// Mitsubishi GX Works2 project: Step Control   PLC: Q01U

PROGRAM conveyor
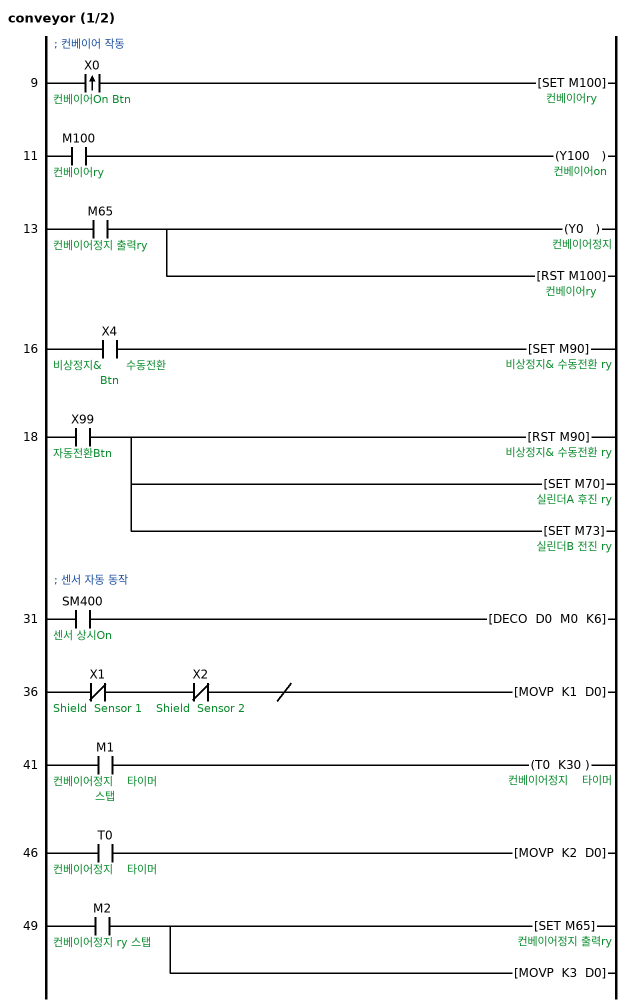
; 컨베이어 작동
9     LDP     X0  ; 컨베이어On Btn
      SET     M100  ; 컨베이어ry
11    LD      M100  ; 컨베이어ry
      OUT     Y100  ; 컨베이어on
13    LD      M65  ; 컨베이어정지 출력ry
      OUT     Y0  ; 컨베이어정지
      RST     M100  ; 컨베이어ry
16    LD      X4  ; 비상정지&       수동전환 Btn
      SET     M90  ; 비상정지& 수동전환 ry
18    LD      X99  ; 자동전환Btn
      RST     M90  ; 비상정지& 수동전환 ry
      SET     M70  ; 실린더A 후진 ry
      SET     M73  ; 실린더B 전진 ry
; 센서 자동 동작
31    LD      SM400  ; 센서 상시On
      DECO    D0 M0 K6
36    LDI     X1  ; Shield  Sensor 1
      ANI     X2  ; Shield  Sensor 2
      INV
      MOVP    K1 D0
41    LD      M1  ; 컨베이어정지    타이머  스탭
      OUT     T0 K30  ; 컨베이어정지    타이머
46    LD      T0  ; 컨베이어정지    타이머
      MOVP    K2 D0
49    LD      M2  ; 컨베이어정지 ry 스탭
      SET     M65  ; 컨베이어정지 출력ry
      MOVP    K3 D0
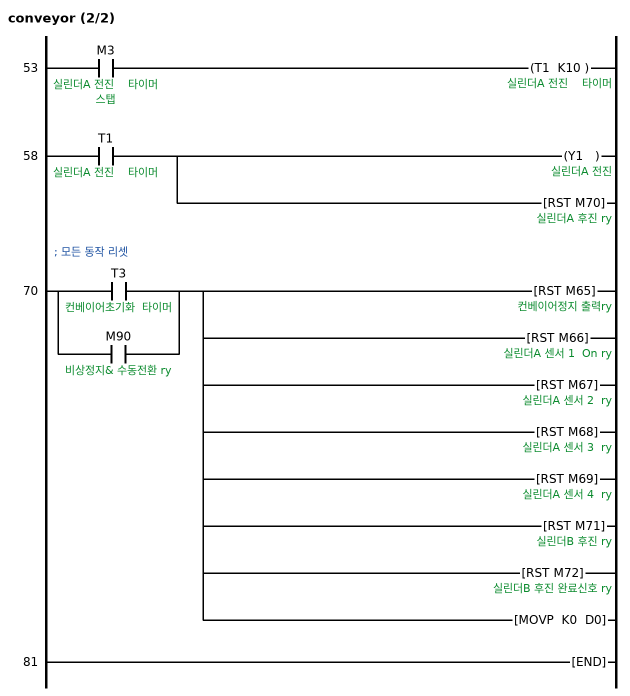
53    LD      M3  ; 실린더A 전진    타이머  스탭
      OUT     T1 K10  ; 실린더A 전진    타이머
58    LD      T1  ; 실린더A 전진    타이머
      OUT     Y1  ; 실린더A 전진
      RST     M70  ; 실린더A 후진 ry
; 모든 동작 리셋
70    LD      T3  ; 컨베이어초기화  타이머
      OR      M90  ; 비상정지& 수동전환 ry
      RST     M65  ; 컨베이어정지 출력ry
      RST     M66  ; 실린더A 센서 1  On ry
      RST     M67  ; 실린더A 센서 2  ry
      RST     M68  ; 실린더A 센서 3  ry
      RST     M69  ; 실린더A 센서 4  ry
      RST     M71  ; 실린더B 후진 ry
      RST     M72  ; 실린더B 후진 완료신호 ry
      MOVP    K0 D0
81    END
END_PROGRAM

PROGRAM cylinder
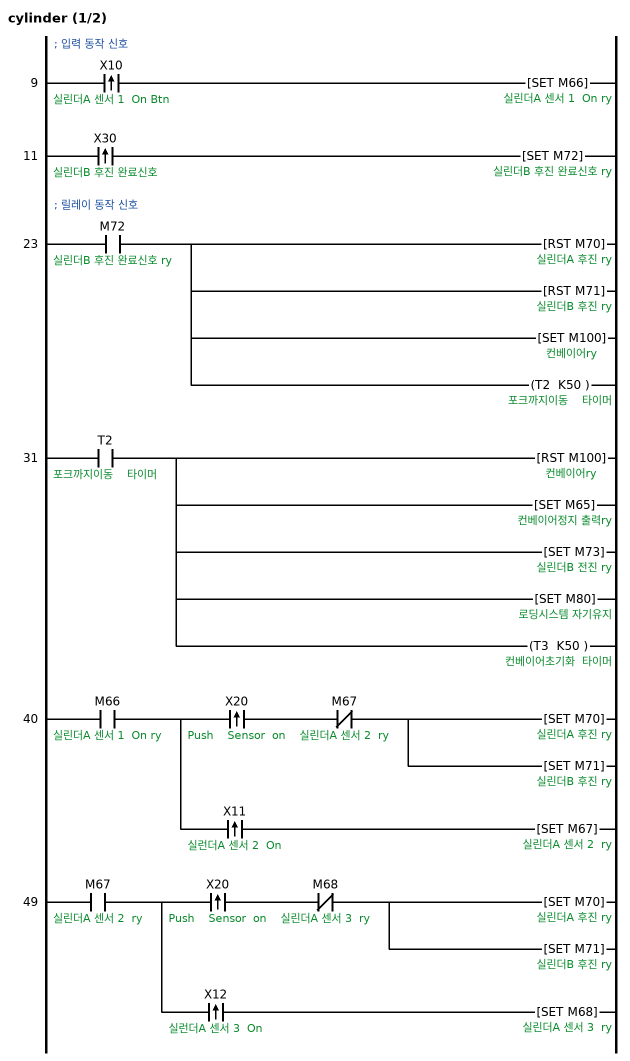
; 입력 동작 신호
9     LDP     X10  ; 실린더A 센서 1  On Btn
      SET     M66  ; 실린더A 센서 1  On ry
11    LDP     X30  ; 실린더B 후진 완료신호
      SET     M72  ; 실린더B 후진 완료신호 ry
; 릴레이 동작 신호
23    LD      M72  ; 실린더B 후진 완료신호 ry
      RST     M70  ; 실린더A 후진 ry
      RST     M71  ; 실린더B 후진 ry
      SET     M100  ; 컨베이어ry
      OUT     T2 K50  ; 포크까지이동    타이머
31    LD      T2  ; 포크까지이동    타이머
      RST     M100  ; 컨베이어ry
      SET     M65  ; 컨베이어정지 출력ry
      SET     M73  ; 실린더B 전진 ry
      SET     M80  ; 로딩시스템 자기유지
      OUT     T3 K50  ; 컨베이어초기화  타이머
40    LD      M66  ; 실린더A 센서 1  On ry
      MPS
      ANDP    X20  ; Push    Sensor  on
      ANI     M67  ; 실린더A 센서 2  ry
      SET     M70  ; 실린더A 후진 ry
      SET     M71  ; 실린더B 후진 ry
      MPP
      ANDP    X11  ; 실런더A 센서 2  On
      SET     M67  ; 실린더A 센서 2  ry
49    LD      M67  ; 실린더A 센서 2  ry
      MPS
      ANDP    X20  ; Push    Sensor  on
      ANI     M68  ; 실린더A 센서 3  ry
      SET     M70  ; 실린더A 후진 ry
      SET     M71  ; 실린더B 후진 ry
      MPP
      ANDP    X12  ; 실런더A 센서 3  On
      SET     M68  ; 실린더A 센서 3  ry
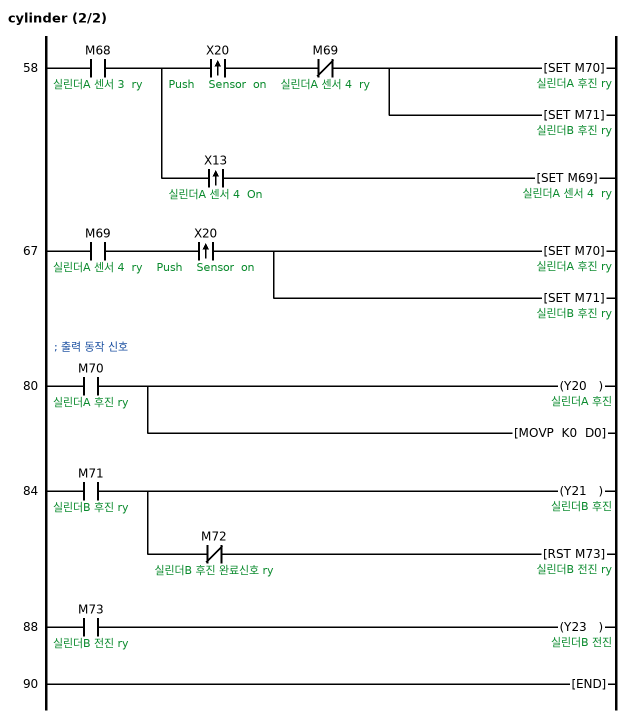
58    LD      M68  ; 실린더A 센서 3  ry
      MPS
      ANDP    X20  ; Push    Sensor  on
      ANI     M69  ; 실린더A 센서 4  ry
      SET     M70  ; 실린더A 후진 ry
      SET     M71  ; 실린더B 후진 ry
      MPP
      ANDP    X13  ; 실린더A 센서 4  On
      SET     M69  ; 실린더A 센서 4  ry
67    LD      M69  ; 실린더A 센서 4  ry
      ANDP    X20  ; Push    Sensor  on
      SET     M70  ; 실린더A 후진 ry
      SET     M71  ; 실린더B 후진 ry
; 출력 동작 신호
80    LD      M70  ; 실린더A 후진 ry
      OUT     Y20  ; 실린더A 후진
      MOVP    K0 D0
84    LD      M71  ; 실린더B 후진 ry
      OUT     Y21  ; 실린더B 후진
      ANI     M72  ; 실린더B 후진 완료신호 ry
      RST     M73  ; 실린더B 전진 ry
88    LD      M73  ; 실린더B 전진 ry
      OUT     Y23  ; 실린더B 전진
90    END
END_PROGRAM

PROGRAM manual
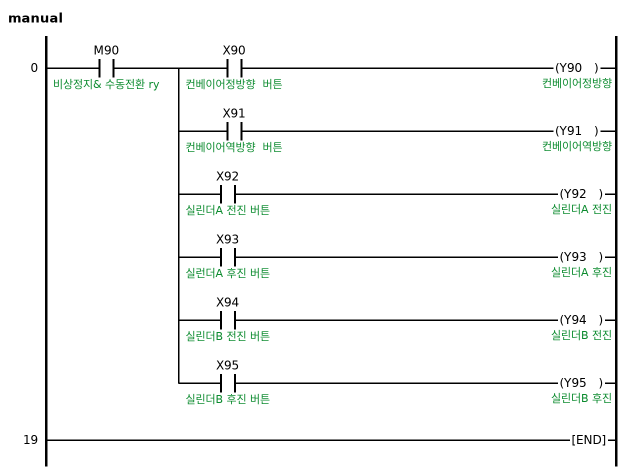
0     LD      M90  ; 비상정지& 수동전환 ry
      MPS
      AND     X90  ; 컨베이어정방향  버튼
      OUT     Y90  ; 컨베이어정방향
      MRD
      AND     X91  ; 컨베이어역방향  버튼
      OUT     Y91  ; 컨베이어역방향
      MRD
      AND     X92  ; 실린더A 전진 버튼
      OUT     Y92  ; 실린더A 전진
      MRD
      AND     X93  ; 실런더A 후진 버튼
      OUT     Y93  ; 실린더A 후진
      MRD
      AND     X94  ; 실린더B 전진 버튼
      OUT     Y94  ; 실린더B 전진
      MPP
      AND     X95  ; 실린더B 후진 버튼
      OUT     Y95  ; 실린더B 후진
19    END
END_PROGRAM

PROGRAM boxSize
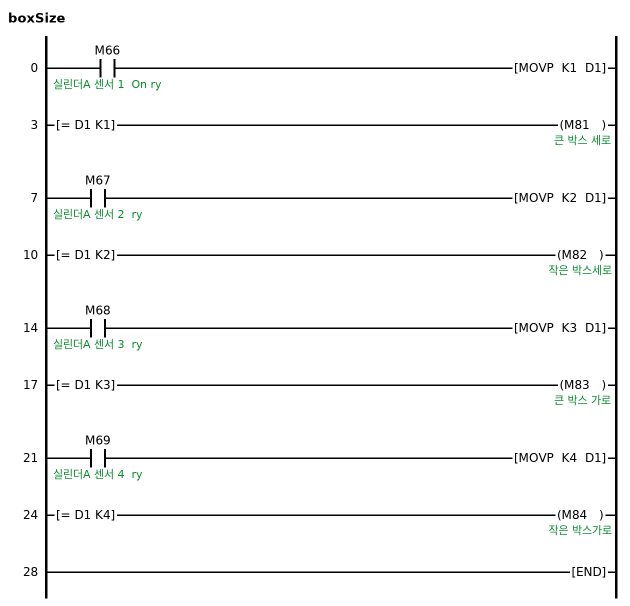
0     LD      M66  ; 실린더A 센서 1  On ry
      MOVP    K1 D1
3     LD=     D1 K1
      OUT     M81  ; 큰 박스 세로
7     LD      M67  ; 실린더A 센서 2  ry
      MOVP    K2 D1
10    LD=     D1 K2
      OUT     M82  ; 작은 박스세로
14    LD      M68  ; 실린더A 센서 3  ry
      MOVP    K3 D1
17    LD=     D1 K3
      OUT     M83  ; 큰 박스 가로
21    LD      M69  ; 실린더A 센서 4  ry
      MOVP    K4 D1
24    LD=     D1 K4
      OUT     M84  ; 작은 박스가로
28    END
END_PROGRAM
